{attribute 'GeneratedUsingTerminal: ELX3252-0000-0016'}
{attribute addProperty BoxType "ELX3252-0000-0016"}
{attribute addProperty Id "StatusAT %I*Status_AE4D73AB5ValueAT %I*INT2"}
{attribute addProperty CRC "1024054797"}
{attribute addProperty Size "7"}
TYPE AI_Standard_Channel_3D09D60D :
STRUCT
	{attribute addProperty Name "Status"}
	Status AT %I* : Status_AE4D73AB;
	{attribute addProperty Name "Value"}
	Value AT %I* : INT;
END_STRUCT
END_TYPE

(* stored: Version 1.2.0.0, ProductVersion 3.1.4024.9
   DUT AI_Standard_Channel_3D09D60D: Id {3f2fb158-9d65-4da4-9fab-8e6da9b7a767} *)
